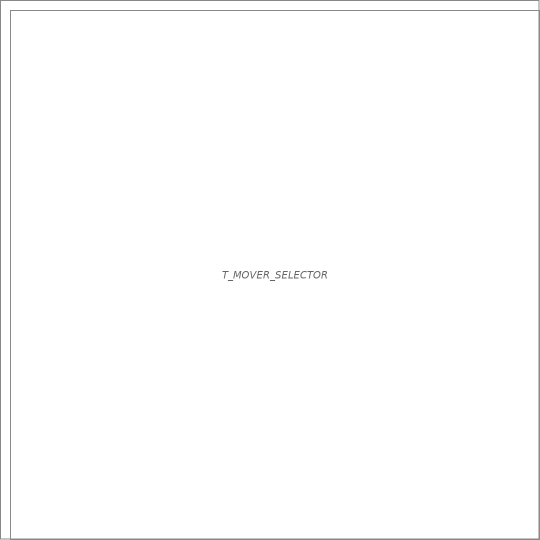
VISUALIZATION SELECTOR_VISU  // 540x540
    Frame (10,10 530x530)
        shows T_MOVER_SELECTOR(Control := GVL_XTS.SelectorCtrl, State := GVL_XTS.SelectorState, sState := MAIN.sSelectorState, sResult := MAIN.sSelectorResult)
END_VISUALIZATION

(* stored: Version 1.1.0.1
   Visu SELECTOR_VISU: Id {e9505c66-7e20-437e-9859-be1cb953ae7b} *)
